FUNCTION_BLOCK PUBLIC ABSTRACT FB_FunctionBase EXTENDS FB_Base
VAR_INPUT
	bSafetyOk	: BOOL 		:= TRUE 				; // Module can operate safely [default true]
END_VAR
VAR_OUTPUT
	sActiveState	: STRING 		:= 'Idle'	; // active state of device 
	bManual			: BOOL 			:= FALSE 	; // device is in manual mode
	bIsSafe			: BOOL 			:= FALSE	; // Device is locked and safe
	bBlockedCommand	: BOOL 			:= FALSE 	; // a device command is blocked because of collision detect 
END_VAR
VAR
	bCmdManual 		: BOOL			:= FALSE	; // manual commands enabled control functions (thus disable automatic)
END_VAR

SUPER^(refFbFault := refFbFault);

// Communicate active state
IF NOT bSafetyOk THEN 
	sActiveState := 'Safety not ok';
ELSIF bErrorActive THEN 
	sActiveState := TO_STRING(stFault.Discription);
ELSIF NOT bInitOk THEN 
	sActiveState := 'Not initialized';
ELSIF bManual THEN 
	sActiveState := 'Operational';
END_IF 

// check for manual command mode
bManual := bCmdManual ;

// Execute device functions
IF bInitOk THEN  
	ExecMachineSafety();
	ExecDevFunctions();
END_IF

// Set fault if commands are blocked
IF bBlockedCommand THEN 
	stFault.Active 			:= TRUE ;
	stFault.ComponentType 	:= E_ComponentTypes.Assembly ;
	stFault.Discription		:= CONCAT( STR1 := sName, STR2 := 'function is blocked');
	stFault.FaultType		:= E_FaultTypes.MC;
END_IF

METHOD PUBLIC CmdManual : BOOL
VAR_INPUT
END_VAR
bCmdManual := true ;
END_METHOD

METHOD PROTECTED ExecDevFunctions : BOOL
VAR_INPUT
END_VAR
END_METHOD

METHOD PRIVATE ExecMachineSafety : BOOL
VAR_INPUT
END_VAR
END_METHOD

END_FUNCTION_BLOCK

(* stored: Version 1.1.0.1, ProductVersion 3.1.4024.5
   POU FB_FunctionBase: Id {ef86906a-1986-411c-841b-bedecc286c14}, SpecialFunc None
   Method CmdManual: Id {a80209b9-b449-43b8-997f-3d83541a6746}
   Method ExecDevFunctions: Id {351765c3-accd-4b4a-927f-08fd149221ad}
   Method ExecMachineSafety: Id {21d44c79-19d0-4d2a-975d-6d59086163c6} *)
